// TwinCAT 3 PLC project TimesTests
// ProgramVersion: 3.1.4024.0
// libraries:
//   Tc2_Standard, * (Beckhoff Automation GmbH)
//   Tc2_System, * (Beckhoff Automation GmbH)
//   Tc3_Module, * (Beckhoff Automation GmbH)
//   TcUnit, * (www.tcunit.org)
//   Times, * (TomasRompotl)
// project tree:
//   Clocks/ PeriodicTriggerTest.TcPOU
//   Convert/ ConvertFunctionsTest.TcPOU
//   / PRG_Test.TcPOU, PlcTask.TcTTO
// (motion and I/O tree: see PLC project types)
// real-time tasks:
//   TASK BindingTestTask: cycle T#1ms, priority 20, ADS port 350
//   TASK PlcTask: cycle T#1ms, priority 21, ADS port 351
//   TASK PlcTask1: cycle T#1ms, priority 22, ADS port 352
//   TASK PlcTask2: cycle T#1ms, priority 23, ADS port 353
//   TASK MathTestTask: cycle T#1ms, priority 24, ADS port 354
//   TASK TimesTestsTask: cycle T#1ms, priority 25, ADS port 355

CONFIGURATION TimesTests
    RESOURCE PLC ON TwinCAT3
        TASK PlcTask(INTERVAL := T#1ms, PRIORITY := 25);
        PROGRAM PRG_Test WITH PlcTask : PRG_Test;
    END_RESOURCE
END_CONFIGURATION

// ---- PRG_Test.TcPOU
PROGRAM PRG_Test
VAR
	convertFunctionsTest : ConvertFunctionsTest();
	periodicTriggerTest : PeriodicTriggerTest();
END_VAR

TcUnit.RUN();

END_PROGRAM

// ---- Convert/ConvertFunctionsTest.TcPOU
FUNCTION_BLOCK ConvertFunctionsTest EXTENDS FB_TestSuite
VAR
END_VAR

SecondsToTimeFunction();
TimeToSecondsFunction();

METHOD SecondsToTimeFunction
VAR_INPUT
END_VAR
TcUnit.TEST('SecondsToTime function');

AssertEquals_TIME(
	Expected := T#5S,
	Actual := SecondsToTime(5),
	Message := 'Converted time is not correct'
);

TEST_FINISHED();
END_METHOD

METHOD TimeToSecondsFunction
VAR_INPUT
END_VAR
TcUnit.TEST('TimeToSeconds function');

AssertEquals_LREAL(
	Expected := 5,
	Actual := TimeToSeconds(T#5S),
	Delta := 0,
	Message := 'Converted seconds are not correct'
);

TEST_FINISHED();
END_METHOD

END_FUNCTION_BLOCK

// ---- Clocks/PeriodicTriggerTest.TcPOU
FUNCTION_BLOCK PeriodicTriggerTest EXTENDS FB_TestSuite
VAR
END_VAR

KeepDisabled();
TriggerWith10msPeriod();

METHOD KeepDisabled
VAR
END_VAR
VAR_INST
	pt : PeriodicTrigger := (Enable := FALSE, Period := T#200MS);
	timer : TON := (IN := TRUE, PT := T#1S);
	wasOn : BOOL;
END_VAR
TcUnit.TEST('Keep disabled');

pt.Cyclic();
wasOn S= pt.Trigger;

timer();
IF (timer.Q) THEN
	timer.IN := FALSE;
	
	AssertEquals_BOOL(
		Expected := FALSE,
		Actual := wasOn,
		Message := 'Periodic trigger triggered when not enabled.'
	);
	
	TEST_FINISHED();
END_IF
END_METHOD

// Test has to be run with 1 ms cycle time
METHOD TriggerWith10msPeriod
VAR
END_VAR
VAR_INST
	pt : PeriodicTrigger := (Enable := TRUE, Period := T#10MS);
	expected : ARRAY[0..40] OF BOOL;
	actual : ARRAY[0..40] OF BOOL;
	cycle : INT := 0;
	init : BOOL := TRUE;
END_VAR
VAR CONSTANT
	EndCycle : INT := 40;
END_VAR
TcUnit.TEST('Trigger with 10 ms period');

IF (init) THEN
	init := FALSE;
	expected[10] := TRUE;
	expected[20] := TRUE;
	expected[30] := TRUE;
END_IF

pt.Cyclic();

IF (cycle < EndCycle) THEN 
	actual[cycle] := pt.Trigger;
	cycle := cycle + 1;

	IF (cycle = EndCycle) THEN
		
		AssertArrayEquals_BOOL(
			Expecteds := expected,
			Actuals := actual,
			Message := 'Periodic trigger should trigger at start of each period after the starting one.'
		);
		
		TEST_FINISHED();
	END_IF
END_IF
END_METHOD

END_FUNCTION_BLOCK
